{attribute 'qualified_only'}
//{attribute 'strict'}
{attribute 'to_string'}
TYPE E_LogicFunction :
(
	OUTPUT := 0,
	REGISTER := 1,
	JUMP := 2,
	CNTUP := 3,
	CNTDN := 4,
	CNTRST := 5,
	NOP := 6,
	CALL := 7
);
END_TYPE

(* stored: Version 1.1.0.1
   EnumerationTextList E_LogicFunction: Id {d239b1bf-4938-4fd9-a1b3-5920e691880e} *)
